(* IEC 61131-3 sources: ArfBotOS/Codesys-4/ArfBotOS.fbsdev/Application.iecapp^/FUN/tcp/FB_PythonServerHandler.fb.st^/public, 3 files *)

(* ---- M_Cancel.meth.st ---- *)
METHOD PUBLIC M_Cancel : BOOL
VAR_INPUT
END_VAR

IF _WorkerUid <> '' THEN
	M_Cancel := TRUE;
	_Command := 'kill: ';
	_Command := CONCAT(_Command, _WorkerUid);
	_WorkerUid := ''; // lets make sure to forget this uid in case its used again for something else
	_Step := 0;
	_Execute := TRUE;

ELSE
	M_Cancel := FALSE;

END_IF
END_METHOD

(* ---- M_Reconnect.meth.st ---- *)
METHOD PUBLIC M_Reconnect : BOOL
VAR_INPUT
END_VAR

_TcpClient._M_Reconnect();
END_METHOD

(* ---- M_Reset.meth.st ---- *)
METHOD PUBLIC M_Reset : BOOL
VAR_INPUT
END_VAR

_Reset := TRUE;
_Error := FALSE;
_ErrorDescription := '';
END_METHOD
